// TIA Portal V17 export
// export: Created 2021-09-08T12:46:16.1780561Z, ExportSetting WithDefaults, DisplayName Totally Integrated Automation Portal, DisplayVersion V17, DisplayName TIA Portal Openness, DisplayVersion V17, DisplayName TIA Portal Version Control Interface, DisplayVersion V17, DisplayName STEP 7 Professional, DisplayVersion V17, DisplayName STEP 7 Safety, DisplayVersion V17, DisplayName WinCC Advanced, DisplayVersion V17
DATA_BLOCK "Data"   // DB10
{ S7_Optimized_Access := 'FALSE' }
VERSION : 1.1
// stored: AutoNumber true, DBAccessibleFromOPCUA true, IsOnlyStoredInLoadMemory false, IsWriteProtectedInAS false
   VAR RETAIN
      Meter1 : Real := 100;   // Inlet water consumption Meter1
   END_VAR
BEGIN
END_DATA_BLOCK
